// Mitsubishi GX Works2 project: BacNinhTap2FX3S   PLC: FX3S

// global labels: Global1
VAR_GLOBAL
  VR1 AT D8030 : INT;
  VR2 AT D8031 : INT;
  XXLimitN AT M8344 : BOOL;
  XXLimitP AT M8343 : BOOL;
  XXBusy AT M8340 : BOOL;
  XXInterruptInverse AT M8347 : BOOL;
  XXPos AT D8340 : DINT;
  XXAccelTime AT D8348 : INT;
  XXDecelTime AT D8349 : INT;
  XXPosView AT D0 : DINT;
  XXTarPos AT D2 : DINT;
  XXFeed AT D4 : DINT;
  XXTarR AT M0 : BOOL;
  XXTarRSkip AT D6 : INT;
  XXOn AT M1 : BOOL;
  XXRun AT M2 : BOOL;
  XXDirection AT M3 : BOOL;
  XXMinI AT X000 : BOOL;
  XXMaxI AT X001 : BOOL;
  XXReadyI AT X002 : BOOL;
  XXPulseO AT Y000 : BOOL;
  XXDirectionO AT Y004 : BOOL;
  XXOnO AT Y002 : BOOL;
  Run AT M4 : BOOL;
  RunI AT X003 : BOOL;
  RunStop AT M5 : BOOL;
  RunStopI AT X004 : BOOL;
  RunState AT D7 : INT;
  RunStateNext AT M6 : BOOL;
  AxisState AT D8 : INT;
  AxisStateNext AT M7 : BOOL;
  FoilExtractState AT D9 : INT;
  FoilExtractStateNext AT M8 : BOOL;
  FoilMoveState AT D10 : INT;
  FoilMoveStateNext AT M9 : BOOL;
  FoilExtractDropN AT M10 : BOOL;
  FoilExtractDropNI AT X005 : BOOL;
  FoilExtractDropNTimer AT TC0 : BOOL;
  FoilExtractDropNTimerDelay AT D11 : INT;
  FoilExtractDropP AT M11 : BOOL;
  FoilExtractDropPI AT X006 : BOOL;
  FoilExtractDropPTimer AT TC1 : BOOL;
  FoilExtractDropPTimerDelay AT D12 : INT;
  FoilExtractDrop AT M12 : BOOL;
  FoilExtractDropO AT Y001 : BOOL;
  FoilExtractFloorN AT M13 : BOOL;
  FoilExtractFloorNI AT X007 : BOOL;
  FoilExtractFloorNTimer AT TC2 : BOOL;
  FoilExtractFloorNTimerDelay AT D13 : INT;
  FoilExtractFloorP AT M14 : BOOL;
  FoilExtractFloorPI AT X010 : BOOL;
  FoilExtractFloorPTimer AT TC3 : BOOL;
  FoilExtractFloorPTimerDelay AT D14 : INT;
  FoilExtractFloor AT M15 : BOOL;
  FoilExtractFloorO AT Y003 : BOOL;
  FoilMoveClampN AT M16 : BOOL;
  FoilMoveClampNTimer AT TC4 : BOOL;
  FoilMoveClampP AT M17 : BOOL;
  FoilMoveClampPTimer AT TC5 : BOOL;
  FoilMoveClampTimerDelay AT D15 : INT;
  FoilMoveClamp AT M18 : BOOL;
  FoilMoveClampO AT Y005 : BOOL;
  FoilMoveSpinN AT M19 : BOOL;
  FoilMoveSpinNI AT X011 : BOOL;
  FoilMoveSpinNTimer AT TC6 : BOOL;
  FoilMoveSpinP AT M20 : BOOL;
  FoilMoveSpinPI AT X012 : BOOL;
  FoilMoveSpinPTimer AT TC7 : BOOL;
  FoilMoveSpinTimerDelay AT D16 : INT;
  FoilMoveSpin AT M21 : BOOL;
  FoilMoveSpinO AT Y006 : BOOL;
  WorkFeed AT D17 : DINT;
END_VAR

// task Task_01 (event TRUE, interval 0, priority 31): POU_01

PROGRAM POU_01
VAR
  fTmp : BOOL;
END_VAR
RST(M8002, XXOn);
MOV(M8002, 200, XXAccelTime);
MOV(M8002, 200, XXDecelTime);
SET(M8002, FoilExtractDrop);
RST(M8002, FoilExtractFloor);
RST(M8002, FoilMoveClamp);
RST(M8002, FoilMoveSpin);
(*1000 pulse = 1 mm, 1 round = 1.75mm, -> servo ppr = 1750*)
DMOV(M8002, (1750 * 2000) / 60, WorkFeed);
(*|||||||||||||||*)
(*|||||||||||||||*)
SET(Run AND RunState = 0, fTmp);
RST(fTmp, Run);
SET(fTmp, XXOn);
MOV(fTmp, 1, RunState);
RST(fTmp, fTmp);
SET(RunStop, fTmp);
RST(fTmp, Run);
RST(fTmp, RunStop);
ZRST(fTmp, RunState, FoilMoveState);
RST(fTmp, XXRun);
SET(fTmp, FoilExtractDrop);
RST(fTmp, FoilExtractFloor);
RST(fTmp, fTmp);
(*|||||||||||||||*)
(*|||||||||||||||*)
INC(RunStateNext, RunState);
INC(AxisStateNext, AxisState);
INC(FoilExtractStateNext, FoilExtractState);
INC(FoilMoveStateNext, FoilMoveState);
ZRST(M8000, RunStateNext, FoilMoveStateNext);
DECO(M8000, RunState, 6, M100);
DECO(M8000, AxisState, 6, M200); DECO(M8000, AxisState, 6, M1200); ZRST(NOT XXTarR OR NOT XXReadyI, M1200, M1263);
DECO(M8000, FoilExtractState, 6, M300);
DECO(M8000, FoilMoveState, 6, M400);
(*|||||||||||||||*)

(*MAIN |||||||||||||||*)
(*origin*)
MOV(M101, 1, AxisState);
MOV(M101, 1, FoilExtractState);
MOV(M101, 1, FoilMoveState);
SET(M101, RunStateNext);
(*ready done, wait run command*)
SET(M102 AND Run, RunStateNext);
(*------cycle step 1*)
SET(M103 AND M1220 AND M330 AND M430, RunStateNext);
(*clamp on*)
MOV(M104, 11, FoilMoveState);
SET(M104, RunStateNext);
(*------cycle step 2*)
SET(M105 AND M415, RunStateNext);
(*tap, extract floor up*)
MOV(M106, 11, AxisState);
MOV(M106, 11, FoilExtractState);
SET(M106, RunStateNext);
(*-----cycle step 3*)
SET(M107 AND M1220 AND M315, RunStateNext);
(*clamp off*)
MOV(M108, 16, FoilMoveState);
SET(M108, RunStateNext);
(*-----cycle step 4*)
SET(M109 AND M420, RunStateNext);
(*extract drop*)
MOV(M110, 16, FoilExtractState);
SET(M110, RunStateNext);
(*-----cycle step 5*)
SET(M111 AND M320, RunStateNext);
(*clamp on*)
MOV(M112, 11, FoilMoveState);
SET(M112, RunStateNext);
(*-----cycle step 6*)
SET(M113 AND M415, RunStateNext);
(*extract floor down*)
MOV(M114, 21, FoilExtractState);
SET(M114, RunStateNext);
(*-----cycle step 7*)
SET(M115 AND M330, RunStateNext);
(*spin*)
MOV(M116, 21, FoilMoveState);
SET(M116, RunStateNext);
(*-----cycle step 8, back to cycle step 1*)
MOV(M117 AND M430, 3, RunState);
(*|||||||||||||||*)

(*AXIS|||||||||||||||*)
(*/////get origin*)
(*at min, jump to move down*)
SET(M1201 AND XXMinI, fTmp);
MOV(fTmp, 3, AxisState); RST(fTmp, fTmp);
(*not at min, move up*)
SET(M1201 AND NOT XXMinI, fTmp);
RST(fTmp, XXPos);
DMOV(fTmp, -60_000, XXTarPos);
DMOV(fTmp, 5_000, XXFeed);
SET(fTmp, XXRun);
SET(fTmp, AxisStateNext); RST(fTmp, fTmp);
(*move up hit limit, reset*)
SET(M202 AND NOT XXBusy, fTmp);
RST(fTmp, XXRun);
RST(fTmp, XXPos);
SET(fTmp, AxisStateNext); RST(fTmp, fTmp);
(*move down*)
SET(M1203, fTmp);
DMOV(fTmp, 5_000, XXTarPos);
DMOV(fTmp, 1_000, XXFeed);
SET(fTmp, XXRun);
SET(fTmp, AxisStateNext); RST(fTmp, fTmp);
(*move down out min, stop*)
SET(M204 AND NOT XXMinI, fTmp);
RST(fTmp, XXRun);
SET(fTmp, AxisStateNext); RST(fTmp, fTmp);
(*stop done, move down 1mm*)
SET(M1205, fTmp);
DMOV(fTmp, XXPos + 1000, XXTarPos);
DMOV(fTmp, 1000, XXFeed);
SET(fTmp, XXRun);
SET(fTmp, AxisStateNext); RST(fTmp, fTmp);
(*move down 1mm done, ready*)
SET(M1206, fTmp);
RST(fTmp, XXPos);
MOV(fTmp, 20, AxisState); RST(fTmp, fTmp);
(*/////main sequence*)
(*wait run hit, move down*)
SET(M1211, fTmp);
DMOV(fTmp, 40_000, XXTarPos);
DMOV(fTmp, WorkFeed, XXFeed);
SET(fTmp, XXRun);
SET(fTmp, AxisStateNext); RST(fTmp, fTmp);
(*target reach or touch max, reset*)
SET(M1212 OR (M212 AND NOT XXBusy), fTmp);
RST(fTmp, XXRun);
SET(fTmp, AxisStateNext); RST(fTmp, fTmp);
(*move down slow done, move up*)
SET(M1213, fTmp);
DMOV(fTmp, 0, XXTarPos);
DMOV(fTmp, WorkFeed, XXFeed);
SET(fTmp, XXRun);
SET(fTmp, AxisStateNext); RST(fTmp, fTmp);
(*move up done, return wait tap hit*)
SET(M1214, fTmp);
MOV(fTmp, 20, AxisState); RST(fTmp, fTmp);
(*|||||||||||||||*)

(*FOIL EXTRACT|||||||||||||||*)
(*get origin*)
SET(M301, FoilExtractDrop);
RST(M301, FoilExtractFloor);
SET(M301 AND FoilExtractDropP AND FoilExtractFloorN, FoilExtractStateNext);
(*get origin done*)
MOV(M302, 30, FoilExtractState);
(*/////floor up*)
(*floor up*)
SET(M311, FoilExtractFloor);
SET(M311 AND FoilExtractFloorP, FoilExtractStateNext);
(**)
MOV(M312, 15, FoilExtractState);
(*/////drop*)
(*drop back*)
RST(M316, FoilExtractDrop);
SET(M316 AND FoilExtractDropN, FoilExtractStateNext);
(*drop forward*)
SET(M317, FoilExtractDrop);
SET(M317 AND FoilExtractDropP, FoilExtractStateNext);
(**)
MOV(M318, 20, FoilExtractState);
(*/////floor down*)
(*floor down*)
RST(M321, FoilExtractFloor);
SET(M321 AND FoilExtractFloorN, FoilExtractStateNext);
(**)
MOV(M322, 30, FoilExtractState);
(*|||||||||||||||*)

(*FOIL MOVE|||||||||||||||*)
(*get origin*)
RST(M401, FoilMoveClamp);
SET(M401 AND FoilMoveClampN, FoilMoveStateNext);
(*get origin done*)
MOV(M402, 30, FoilMoveState);
(*/////clamp*)
(*clamp on*)
SET(M411, FoilMoveClamp);
SET(M411 AND FoilMoveClampP, FoilMoveStateNext);
(**)
MOV(M412, 15, FoilMoveState);
(*clamp off*)
RST(M416, FoilMoveClamp);
SET(M416 AND FoilMoveClampN, FoilMoveStateNext);
(**)
MOV(M417, 20, FoilMoveState);
(*/////spin*)
(*spin*)
MOV(M421 AND FoilMoveSpin, 22, FoilMoveState);
MOV(M421 AND NOT FoilMoveSpin, 26, FoilMoveState);
(*spin rst*)
RST(M422, FoilMoveSpin);
SET(M422 AND FoilMoveSpinN, FoilMoveStateNext);
(*end*)
MOV(M423, 30, FoilMoveState);
(*spin set*)
SET(M426, FoilMoveSpin);
SET(M426 AND FoilMoveSpinP, FoilMoveStateNext);
(*end*)
MOV(M427, 30, FoilMoveState);

(*|||||||||||||||*)
(*XX*)
RST(XXRun AND XXTarPos = XXPos, XXRun);
DDRVA(XXRun, XXTarPos, XXFeed, XXPulseO, XXDirection);
RST(M8029, XXRun);
OUT(XXDirection, XXDirectionO);
INC(NOT XXRun AND NOT XXBusy AND XXTarRSkip < 5, XXTarRSkip);
RST(XXRun, XXTarRSkip);
OUT(XXTarRSkip >= 5, XXTarR);
(**)
OUT(XXMinI, XXLimitN);
OUT(XXMaxI, XXLimitP);
(*|||||||||||||||*)

MOV(M8000, 1 + (VR1 / 16), FoilExtractDropNTimerDelay);
MOV(M8000, 1 + (VR2 / 16), FoilMoveSpinTimerDelay);
(*|||||||||||||||*)
PLS(RunI, Run); SET(Run, Run);
PLS(RunStopI, RunStop); SET(RunStop, RunStop);
OUT_T(NOT FoilExtractDrop, FoilExtractDropNTimer, FoilExtractDropNTimerDelay); SET(FoilExtractDropNTimer, FoilExtractDropN); RST(FoilExtractDropNTimer, FoilExtractDropP);
OUT_T(FoilExtractDrop, FoilExtractDropPTimer, 1); SET(FoilExtractDropPTimer, FoilExtractDropP); RST(FoilExtractDropPTimer, FoilExtractDropN);
OUT_T(FoilExtractFloorNI, FoilExtractFloorNTimer, 1); SET(FoilExtractFloorNTimer, FoilExtractFloorN); RST(FoilExtractFloorNTimer, FoilExtractFloorP);
OUT_T(FoilExtractFloorPI, FoilExtractFloorPTimer, 1); SET(FoilExtractFloorPTimer, FoilExtractFloorP); RST(FoilExtractFloorPTimer, FoilExtractFloorN);
OUT_T(NOT FoilMoveClamp, FoilMoveClampNTimer, 3); SET(FoilMoveClampNTimer, FoilMoveClampN); RST(FoilMoveClampNTimer, FoilMoveClampP);
OUT_T(FoilMoveClamp, FoilMoveClampPTimer, 3); SET(FoilMoveClampPTimer, FoilMoveClampP); RST(FoilMoveClampPTimer, FoilMoveClampN);
OUT_T(FoilMoveSpinNI, FoilMoveSpinNTimer, FoilMoveSpinTimerDelay); SET(FoilMoveSpinNTimer, FoilMoveSpinN); RST(FoilMoveSpinNTimer, FoilMoveSpinP);
OUT_T(FoilMoveSpinPI, FoilMoveSpinPTimer, FoilMoveSpinTimerDelay); SET(FoilMoveSpinPTimer, FoilMoveSpinP); RST(FoilMoveSpinPTimer, FoilMoveSpinN);
(*|||||||||||||||*)
OUT(XXOn, XXOnO);
OUT(NOT FoilExtractDrop, FoilExtractDropO);
OUT(FoilExtractFloor, FoilExtractFloorO);
OUT(FoilMoveClamp, FoilMoveClampO);
OUT(FoilMoveSpin, FoilMoveSpinO);
(*|||||||||||||||*)
END_PROGRAM
